{attribute 'qualified_only'}
{attribute 'strict'}
TYPE FeedrateInterpolation :
(
	CONST := Tc2_PlcInterpolation.E_NciFeedRateIpol.E_NciFeedrateIpolConstant,
    LINEAR := Tc2_PlcInterpolation.E_NciFeedRateIpol.E_NciFeedrateIpolLinear
) UINT;
END_TYPE

(* stored: Version 1.1.0.1, ProductVersion 3.1.4024.12
   DUT FeedrateInterpolation: Id {27dd3381-484b-4b89-a6f1-ade266d21be3} *)
